FUNCTION_BLOCK FB_HMI_TEMPERATURES EXTENDS FB_HMI_COMPONENT
VAR_INPUT
END_VAR
VAR_OUTPUT
END_VAR

VAR_IN_OUT
    voters          : FB_METIS_VOTERS;
END_VAR
VAR
    // active tab of the main frame
    eActiveTab : E_HMI_TEMP_TABS := E_HMI_TEMP_TABS.VOTERS;
    sActiveName : STRING;
    
    // components
    fbVoters       		: FB_HMI_TEMP_VOTERS;

    
    // buttons
    fbVotersButton       : FB_HMI_BUTTON(sName := 'Voters'               , sIconName := '', nThisTab := E_HMI_CRY_TABS.VOTERS);

END_VAR

// update the components

fbVoters(fbInstance := voters);

// update the buttons

fbVotersButton(
    stColor     := fbVoters.fbStatusColor,
    nActiveTab  := eActiveTab,
    sActiveName := sActiveName);



// update the summary health/busy status
fbHealthStatus(
    bIsEnabled  := TRUE,
    bIsGood     :=     fbVoters.fbHealthStatus.bGood,
    bHasWarning :=     fbVoters.fbHealthStatus.bWarning);

fbBusyStatus(
    bIsEnabled   := TRUE,
    bIsBusy      :=    fbVoters.fbBusyStatus.bBusy);

M_UpdateStatusColor();

END_FUNCTION_BLOCK

(* stored: Version 1.1.0.1, ProductVersion 3.1.4024.14
   POU FB_HMI_TEMPERATURES: Id {575ff2c9-a964-4186-9084-4c0cc38e6ece}, SpecialFunc None *)
